# EPICS substitutions: ek9000App/Db/EL3024.substitutions
file EL3024.template
{       pattern
        {
                TERMINAL,

        }
        {
        }
}
